// TIA Portal V20 export
ORGANIZATION_BLOCK "Startup"   // OB1015, LAD, Startup
TITLE = "Complete Restart"
// stored: AutoNumber false, IsIECCheckEnabled true, Namespace Unit1.Em2, SetENOAutomatically true
   VAR_INPUT
      LostRetentive : Bool;   // True if retentive data are lost
      LostRTC : Bool;   // True if date and time are lost
   END_VAR
BEGIN

REGION Network 1 (SCL): Build the Absolut Reference Designator
   // Set the Absoult Reference Designator in the Config DB
   IF LEN(IN := "Unit1.Em2.Config".em.referenceDesignator.parent) <> 0 THEN
       "Unit1.Em2.Config".em.referenceDesignator.combined := CONCAT_WSTRING(IN1 := "Unit1.Em2.Config".em.referenceDesignator.parent, IN2 := WSTRING#'.', IN3 := "Unit1.Em2.Config".em.referenceDesignator.relative);
   ELSE
       "Unit1.Em2.Config".em.referenceDesignator.combined := "Unit1.Em2.Config".em.referenceDesignator.relative;
   END_IF;
END_REGION

REGION Network 2 (SCL): CM Config
   // 
   "Unit1.Em2.Config".cmElectrodeFixRightTopFwdBwd .referenceDesignator := WSTRING#'Electrode Fix Right Top';
   "Unit1.Em2.Config".cmElectrodeFixRightTopFwdBwd .monitoringLeavingFeedback := T#5s;
   "Unit1.Em2.Config".cmElectrodeFixRightTopFwdBwd .monitoringReachingFeedback := T#5s;
   "Unit1.Em2.Config".cmElectrodeFixRightTopFwdBwd .monitoringDiscrepancy := T#1s;
   "Unit1.Em2.Config".cmElectrodeFixRightTopFwdBwd .setOutputHomeContinuously := TRUE;
   "Unit1.Em2.Config".cmElectrodeFixRightTopFwdBwd .setOutputWorkContinuously := TRUE;
   "Unit1.Em2.Config".cmElectrodeFixRightTopFwdBwd .disableHomeCommand := FALSE;
   "Unit1.Em2.Config".cmElectrodeFixRightTopFwdBwd .disableFeedbackHomePos := FALSE;
   "Unit1.Em2.Config".cmElectrodeFixRightTopFwdBwd .disableFeedbackWorkPos := FALSE;
   "Unit1.Em2.Config".cmElectrodeFixRightTopFwdBwd .disableAlarms := FALSE;
   "Unit1.Em2.Config".cmElectrodeFixRightTopFwdBwd .resetOutputsOnError := FALSE;
   "Unit1.Em2.Config".cmElectrodeFixRightTopFwdBwd .allwaysWaitOnReachingTime := FALSE;


   // 
   "Unit1.Em2.Config".cmElectrodeFixRightBottomFwdBwd.referenceDesignator := WSTRING#'Electrode Fix Right BTM';
   "Unit1.Em2.Config".cmElectrodeFixRightBottomFwdBwd.monitoringLeavingFeedback := T#5s;
   "Unit1.Em2.Config".cmElectrodeFixRightBottomFwdBwd.monitoringReachingFeedback := T#5s;
   "Unit1.Em2.Config".cmElectrodeFixRightBottomFwdBwd.monitoringDiscrepancy := T#1s;
   "Unit1.Em2.Config".cmElectrodeFixRightBottomFwdBwd.setOutputHomeContinuously := TRUE;
   "Unit1.Em2.Config".cmElectrodeFixRightBottomFwdBwd.setOutputWorkContinuously := TRUE;
   "Unit1.Em2.Config".cmElectrodeFixRightBottomFwdBwd.disableHomeCommand := FALSE;
   "Unit1.Em2.Config".cmElectrodeFixRightBottomFwdBwd.disableFeedbackHomePos := FALSE;
   "Unit1.Em2.Config".cmElectrodeFixRightBottomFwdBwd.disableFeedbackWorkPos := FALSE;
   "Unit1.Em2.Config".cmElectrodeFixRightBottomFwdBwd.disableAlarms := FALSE;
   "Unit1.Em2.Config".cmElectrodeFixRightBottomFwdBwd.resetOutputsOnError := FALSE;
   "Unit1.Em2.Config".cmElectrodeFixRightBottomFwdBwd.allwaysWaitOnReachingTime := FALSE;

   // 
   "Unit1.Em2.Config".cmElectrodeFixLeftTopFwdBwd.referenceDesignator := WSTRING#'Electrode Fix Left Top';
   "Unit1.Em2.Config".cmElectrodeFixLeftTopFwdBwd.monitoringLeavingFeedback := T#5s;
   "Unit1.Em2.Config".cmElectrodeFixLeftTopFwdBwd.monitoringReachingFeedback := T#5s;
   "Unit1.Em2.Config".cmElectrodeFixLeftTopFwdBwd.monitoringDiscrepancy := T#1s;
   "Unit1.Em2.Config".cmElectrodeFixLeftTopFwdBwd.setOutputHomeContinuously := TRUE;
   "Unit1.Em2.Config".cmElectrodeFixLeftTopFwdBwd.setOutputWorkContinuously := TRUE;
   "Unit1.Em2.Config".cmElectrodeFixLeftTopFwdBwd.disableHomeCommand := FALSE;
   "Unit1.Em2.Config".cmElectrodeFixLeftTopFwdBwd.disableFeedbackHomePos := FALSE;
   "Unit1.Em2.Config".cmElectrodeFixLeftTopFwdBwd.disableFeedbackWorkPos := FALSE;
   "Unit1.Em2.Config".cmElectrodeFixLeftTopFwdBwd.disableAlarms := FALSE;
   "Unit1.Em2.Config".cmElectrodeFixLeftTopFwdBwd.resetOutputsOnError := FALSE;
   "Unit1.Em2.Config".cmElectrodeFixLeftTopFwdBwd.allwaysWaitOnReachingTime := FALSE;


   // 
   "Unit1.Em2.Config".cmElectrodeFixLeftBottomFwdBwd.referenceDesignator := WSTRING#'Electrode Fix Left BTM';
   "Unit1.Em2.Config".cmElectrodeFixLeftBottomFwdBwd.monitoringLeavingFeedback := T#5s;
   "Unit1.Em2.Config".cmElectrodeFixLeftBottomFwdBwd.monitoringReachingFeedback := T#5s;
   "Unit1.Em2.Config".cmElectrodeFixLeftBottomFwdBwd.monitoringDiscrepancy := T#1s;
   "Unit1.Em2.Config".cmElectrodeFixLeftBottomFwdBwd.setOutputHomeContinuously := TRUE;
   "Unit1.Em2.Config".cmElectrodeFixLeftBottomFwdBwd.setOutputWorkContinuously := TRUE;
   "Unit1.Em2.Config".cmElectrodeFixLeftBottomFwdBwd.disableHomeCommand := FALSE;
   "Unit1.Em2.Config".cmElectrodeFixLeftBottomFwdBwd.disableFeedbackHomePos := FALSE;
   "Unit1.Em2.Config".cmElectrodeFixLeftBottomFwdBwd.disableFeedbackWorkPos := FALSE;
   "Unit1.Em2.Config".cmElectrodeFixLeftBottomFwdBwd.disableAlarms := FALSE;
   "Unit1.Em2.Config".cmElectrodeFixLeftBottomFwdBwd.resetOutputsOnError := FALSE;
   "Unit1.Em2.Config".cmElectrodeFixLeftBottomFwdBwd.allwaysWaitOnReachingTime := FALSE;


   // 
   "Unit1.Em2.Config".cmElectrodeFixLeftTopUpDown.referenceDesignator := WSTRING#'Electrode Fix Left Top';
   "Unit1.Em2.Config".cmElectrodeFixLeftTopUpDown.monitoringLeavingFeedback := T#5s;
   "Unit1.Em2.Config".cmElectrodeFixLeftTopUpDown.monitoringReachingFeedback := T#5s;
   "Unit1.Em2.Config".cmElectrodeFixLeftTopUpDown.monitoringDiscrepancy := T#1s;
   "Unit1.Em2.Config".cmElectrodeFixLeftTopUpDown.setOutputHomeContinuously := TRUE;
   "Unit1.Em2.Config".cmElectrodeFixLeftTopUpDown.setOutputWorkContinuously := TRUE;
   "Unit1.Em2.Config".cmElectrodeFixLeftTopUpDown.disableHomeCommand := FALSE;
   "Unit1.Em2.Config".cmElectrodeFixLeftTopUpDown.disableFeedbackHomePos := FALSE;
   "Unit1.Em2.Config".cmElectrodeFixLeftTopUpDown.disableFeedbackWorkPos := FALSE;
   "Unit1.Em2.Config".cmElectrodeFixLeftTopUpDown.disableAlarms := FALSE;
   "Unit1.Em2.Config".cmElectrodeFixLeftTopUpDown.resetOutputsOnError := FALSE;
   "Unit1.Em2.Config".cmElectrodeFixLeftTopUpDown.allwaysWaitOnReachingTime := FALSE;


   // 
   "Unit1.Em2.Config".cmElectrodeFixLeftBottomUpDown.referenceDesignator := WSTRING#'Electrode Fix Left BTM';
   "Unit1.Em2.Config".cmElectrodeFixLeftBottomUpDown.monitoringLeavingFeedback := T#5s;
   "Unit1.Em2.Config".cmElectrodeFixLeftBottomUpDown.monitoringReachingFeedback := T#5s;
   "Unit1.Em2.Config".cmElectrodeFixLeftBottomUpDown.monitoringDiscrepancy := T#1s;
   "Unit1.Em2.Config".cmElectrodeFixLeftBottomUpDown.setOutputHomeContinuously := TRUE;
   "Unit1.Em2.Config".cmElectrodeFixLeftBottomUpDown.setOutputWorkContinuously := TRUE;
   "Unit1.Em2.Config".cmElectrodeFixLeftBottomUpDown.disableHomeCommand := FALSE;
   "Unit1.Em2.Config".cmElectrodeFixLeftBottomUpDown.disableFeedbackHomePos := FALSE;
   "Unit1.Em2.Config".cmElectrodeFixLeftBottomUpDown.disableFeedbackWorkPos := FALSE;
   "Unit1.Em2.Config".cmElectrodeFixLeftBottomUpDown.disableAlarms := FALSE;
   "Unit1.Em2.Config".cmElectrodeFixLeftBottomUpDown.resetOutputsOnError := FALSE;
   "Unit1.Em2.Config".cmElectrodeFixLeftBottomUpDown.allwaysWaitOnReachingTime := FALSE;


   // 
   "Unit1.Em2.Config".cmUwSemiSplicerVacuumRightTopOnOff.referenceDesignator := WSTRING#'Splicer Vacuum Right Top';
   "Unit1.Em2.Config".cmUwSemiSplicerVacuumRightTopOnOff.monitoringLeavingFeedback := T#5s;
   "Unit1.Em2.Config".cmUwSemiSplicerVacuumRightTopOnOff.monitoringReachingFeedback := T#1S;
   "Unit1.Em2.Config".cmUwSemiSplicerVacuumRightTopOnOff.monitoringDiscrepancy := T#1s;
   "Unit1.Em2.Config".cmUwSemiSplicerVacuumRightTopOnOff.setOutputHomeContinuously := FALSE;
   "Unit1.Em2.Config".cmUwSemiSplicerVacuumRightTopOnOff.setOutputWorkContinuously := TRUE;
   "Unit1.Em2.Config".cmUwSemiSplicerVacuumRightTopOnOff.disableHomeCommand := FALSE;
   "Unit1.Em2.Config".cmUwSemiSplicerVacuumRightTopOnOff.disableFeedbackHomePos := TRUE;
   "Unit1.Em2.Config".cmUwSemiSplicerVacuumRightTopOnOff.disableFeedbackWorkPos := FALSE;
   "Unit1.Em2.Config".cmUwSemiSplicerVacuumRightTopOnOff.disableAlarms := FALSE;
   "Unit1.Em2.Config".cmUwSemiSplicerVacuumRightTopOnOff.resetOutputsOnError := FALSE;
   "Unit1.Em2.Config".cmUwSemiSplicerVacuumRightTopOnOff.allwaysWaitOnReachingTime := FALSE;


   // 
   "Unit1.Em2.Config".cmUwSemiSplicerVacuumRightBottomOnOff.referenceDesignator := WSTRING#'Splicer Vacuum Right BTM';
   "Unit1.Em2.Config".cmUwSemiSplicerVacuumRightBottomOnOff.monitoringLeavingFeedback := T#5s;
   "Unit1.Em2.Config".cmUwSemiSplicerVacuumRightBottomOnOff.monitoringReachingFeedback := T#1S;
   "Unit1.Em2.Config".cmUwSemiSplicerVacuumRightBottomOnOff.monitoringDiscrepancy := T#1s;
   "Unit1.Em2.Config".cmUwSemiSplicerVacuumRightBottomOnOff.setOutputHomeContinuously := FALSE;
   "Unit1.Em2.Config".cmUwSemiSplicerVacuumRightBottomOnOff.setOutputWorkContinuously := TRUE;
   "Unit1.Em2.Config".cmUwSemiSplicerVacuumRightBottomOnOff.disableHomeCommand := FALSE;
   "Unit1.Em2.Config".cmUwSemiSplicerVacuumRightBottomOnOff.disableFeedbackHomePos := TRUE;
   "Unit1.Em2.Config".cmUwSemiSplicerVacuumRightBottomOnOff.disableFeedbackWorkPos := FALSE;
   "Unit1.Em2.Config".cmUwSemiSplicerVacuumRightBottomOnOff.disableAlarms := FALSE;
   "Unit1.Em2.Config".cmUwSemiSplicerVacuumRightBottomOnOff.resetOutputsOnError := FALSE;
   "Unit1.Em2.Config".cmUwSemiSplicerVacuumRightBottomOnOff.allwaysWaitOnReachingTime := FALSE;


   // 
   "Unit1.Em2.Config".cmUwSemiSplicerVacuumLeftTopOnOff.referenceDesignator := WSTRING#'Splicer Vacuum Left Top';
   "Unit1.Em2.Config".cmUwSemiSplicerVacuumLeftTopOnOff.monitoringLeavingFeedback := T#5s;
   "Unit1.Em2.Config".cmUwSemiSplicerVacuumLeftTopOnOff.monitoringReachingFeedback := T#1S;
   "Unit1.Em2.Config".cmUwSemiSplicerVacuumLeftTopOnOff.monitoringDiscrepancy := T#1s;
   "Unit1.Em2.Config".cmUwSemiSplicerVacuumLeftTopOnOff.setOutputHomeContinuously := FALSE;
   "Unit1.Em2.Config".cmUwSemiSplicerVacuumLeftTopOnOff.setOutputWorkContinuously := TRUE;
   "Unit1.Em2.Config".cmUwSemiSplicerVacuumLeftTopOnOff.disableHomeCommand := FALSE;
   "Unit1.Em2.Config".cmUwSemiSplicerVacuumLeftTopOnOff.disableFeedbackHomePos := TRUE;
   "Unit1.Em2.Config".cmUwSemiSplicerVacuumLeftTopOnOff.disableFeedbackWorkPos := FALSE;
   "Unit1.Em2.Config".cmUwSemiSplicerVacuumLeftTopOnOff.disableAlarms := FALSE;
   "Unit1.Em2.Config".cmUwSemiSplicerVacuumLeftTopOnOff.resetOutputsOnError := FALSE;
   "Unit1.Em2.Config".cmUwSemiSplicerVacuumLeftTopOnOff.allwaysWaitOnReachingTime := FALSE;


   // 
   "Unit1.Em2.Config".cmUwSemiSplicerVacuumLeftBottomOnOff.referenceDesignator := WSTRING#'Splicer Vacuum Left BTM';
   "Unit1.Em2.Config".cmUwSemiSplicerVacuumLeftBottomOnOff.monitoringLeavingFeedback := T#5s;
   "Unit1.Em2.Config".cmUwSemiSplicerVacuumLeftBottomOnOff.monitoringReachingFeedback := T#1S;
   "Unit1.Em2.Config".cmUwSemiSplicerVacuumLeftBottomOnOff.monitoringDiscrepancy := T#1s;
   "Unit1.Em2.Config".cmUwSemiSplicerVacuumLeftBottomOnOff.setOutputHomeContinuously := FALSE;
   "Unit1.Em2.Config".cmUwSemiSplicerVacuumLeftBottomOnOff.setOutputWorkContinuously := TRUE;
   "Unit1.Em2.Config".cmUwSemiSplicerVacuumLeftBottomOnOff.disableHomeCommand := FALSE;
   "Unit1.Em2.Config".cmUwSemiSplicerVacuumLeftBottomOnOff.disableFeedbackHomePos := TRUE;
   "Unit1.Em2.Config".cmUwSemiSplicerVacuumLeftBottomOnOff.disableFeedbackWorkPos := FALSE;
   "Unit1.Em2.Config".cmUwSemiSplicerVacuumLeftBottomOnOff.disableAlarms := FALSE;
   "Unit1.Em2.Config".cmUwSemiSplicerVacuumLeftBottomOnOff.resetOutputsOnError := FALSE;
   "Unit1.Em2.Config".cmUwSemiSplicerVacuumLeftBottomOnOff.allwaysWaitOnReachingTime := FALSE;


   // Electrode Cutter
   "Unit1.Em2.Config".cmElectrodeCutterFwdBwd.referenceDesignator := WSTRING#'Electrode Cutter';
   "Unit1.Em2.Config".cmElectrodeCutterFwdBwd.monitoringLeavingFeedback := T#5s;
   "Unit1.Em2.Config".cmElectrodeCutterFwdBwd.monitoringReachingFeedback := T#5s;
   "Unit1.Em2.Config".cmElectrodeCutterFwdBwd.monitoringDiscrepancy := T#1s;
   "Unit1.Em2.Config".cmElectrodeCutterFwdBwd.setOutputHomeContinuously := TRUE;
   "Unit1.Em2.Config".cmElectrodeCutterFwdBwd.setOutputWorkContinuously := TRUE;
   "Unit1.Em2.Config".cmElectrodeCutterFwdBwd.disableHomeCommand := FALSE;
   "Unit1.Em2.Config".cmElectrodeCutterFwdBwd.disableFeedbackHomePos := FALSE;
   "Unit1.Em2.Config".cmElectrodeCutterFwdBwd.disableFeedbackWorkPos := FALSE;
   "Unit1.Em2.Config".cmElectrodeCutterFwdBwd.disableAlarms := FALSE;
   "Unit1.Em2.Config".cmElectrodeCutterFwdBwd.resetOutputsOnError := FALSE;
   "Unit1.Em2.Config".cmElectrodeCutterFwdBwd.allwaysWaitOnReachingTime := FALSE;


   // 
   "Unit1.Em2.Config".cmSplicingLeftModuleMoverFwdBwd.referenceDesignator := WSTRING#'Left Module Mover';
   "Unit1.Em2.Config".cmSplicingLeftModuleMoverFwdBwd.monitoringLeavingFeedback := T#30s;
   "Unit1.Em2.Config".cmSplicingLeftModuleMoverFwdBwd.monitoringReachingFeedback := T#30s;
   "Unit1.Em2.Config".cmSplicingLeftModuleMoverFwdBwd.monitoringDiscrepancy := T#1s;
   "Unit1.Em2.Config".cmSplicingLeftModuleMoverFwdBwd.setOutputHomeContinuously := TRUE;
   "Unit1.Em2.Config".cmSplicingLeftModuleMoverFwdBwd.setOutputWorkContinuously := TRUE;
   "Unit1.Em2.Config".cmSplicingLeftModuleMoverFwdBwd.disableHomeCommand := FALSE;
   "Unit1.Em2.Config".cmSplicingLeftModuleMoverFwdBwd.disableFeedbackHomePos := FALSE;
   "Unit1.Em2.Config".cmSplicingLeftModuleMoverFwdBwd.disableFeedbackWorkPos := FALSE;
   "Unit1.Em2.Config".cmSplicingLeftModuleMoverFwdBwd.disableAlarms := FALSE;
   "Unit1.Em2.Config".cmSplicingLeftModuleMoverFwdBwd.resetOutputsOnError := FALSE;
   "Unit1.Em2.Config".cmSplicingLeftModuleMoverFwdBwd.allwaysWaitOnReachingTime := FALSE;


   // 
   "Unit1.Em2.Config".cmSplicingRightModuleMoverFwdBwd.referenceDesignator := WSTRING#'Right Module Mover';
   "Unit1.Em2.Config".cmSplicingRightModuleMoverFwdBwd.monitoringLeavingFeedback := T#30s;
   "Unit1.Em2.Config".cmSplicingRightModuleMoverFwdBwd.monitoringReachingFeedback := T#30s;
   "Unit1.Em2.Config".cmSplicingRightModuleMoverFwdBwd.monitoringDiscrepancy := T#1s;
   "Unit1.Em2.Config".cmSplicingRightModuleMoverFwdBwd.setOutputHomeContinuously := TRUE;
   "Unit1.Em2.Config".cmSplicingRightModuleMoverFwdBwd.setOutputWorkContinuously := TRUE;
   "Unit1.Em2.Config".cmSplicingRightModuleMoverFwdBwd.disableHomeCommand := FALSE;
   "Unit1.Em2.Config".cmSplicingRightModuleMoverFwdBwd.disableFeedbackHomePos := FALSE;
   "Unit1.Em2.Config".cmSplicingRightModuleMoverFwdBwd.disableFeedbackWorkPos := FALSE;
   "Unit1.Em2.Config".cmSplicingRightModuleMoverFwdBwd.disableAlarms := FALSE;
   "Unit1.Em2.Config".cmSplicingRightModuleMoverFwdBwd.resetOutputsOnError := FALSE;
   "Unit1.Em2.Config".cmSplicingRightModuleMoverFwdBwd.allwaysWaitOnReachingTime := FALSE;


   // 
   "Unit1.Em2.Config".cmElectrodeLeftHolderMoverFwdBwd.referenceDesignator := WSTRING#'Left Holder Mover';
   "Unit1.Em2.Config".cmElectrodeLeftHolderMoverFwdBwd.monitoringLeavingFeedback := T#5s;
   "Unit1.Em2.Config".cmElectrodeLeftHolderMoverFwdBwd.monitoringReachingFeedback := T#5s;
   "Unit1.Em2.Config".cmElectrodeLeftHolderMoverFwdBwd.monitoringDiscrepancy := T#1s;
   "Unit1.Em2.Config".cmElectrodeLeftHolderMoverFwdBwd.setOutputHomeContinuously := TRUE;
   "Unit1.Em2.Config".cmElectrodeLeftHolderMoverFwdBwd.setOutputWorkContinuously := TRUE;
   "Unit1.Em2.Config".cmElectrodeLeftHolderMoverFwdBwd.disableHomeCommand := FALSE;
   "Unit1.Em2.Config".cmElectrodeLeftHolderMoverFwdBwd.disableFeedbackHomePos := FALSE;
   "Unit1.Em2.Config".cmElectrodeLeftHolderMoverFwdBwd.disableFeedbackWorkPos := FALSE;
   "Unit1.Em2.Config".cmElectrodeLeftHolderMoverFwdBwd.disableAlarms := FALSE;
   "Unit1.Em2.Config".cmElectrodeLeftHolderMoverFwdBwd.resetOutputsOnError := FALSE;
   "Unit1.Em2.Config".cmElectrodeLeftHolderMoverFwdBwd.allwaysWaitOnReachingTime := FALSE;


   // 
   "Unit1.Em2.Config".cmElectrodeRightHolderMoverFwdBwd.referenceDesignator := WSTRING#'Right Holder Mover';
   "Unit1.Em2.Config".cmElectrodeRightHolderMoverFwdBwd.monitoringLeavingFeedback := T#5s;
   "Unit1.Em2.Config".cmElectrodeRightHolderMoverFwdBwd.monitoringReachingFeedback := T#5s;
   "Unit1.Em2.Config".cmElectrodeRightHolderMoverFwdBwd.monitoringDiscrepancy := T#1s;
   "Unit1.Em2.Config".cmElectrodeRightHolderMoverFwdBwd.setOutputHomeContinuously := TRUE;
   "Unit1.Em2.Config".cmElectrodeRightHolderMoverFwdBwd.setOutputWorkContinuously := TRUE;
   "Unit1.Em2.Config".cmElectrodeRightHolderMoverFwdBwd.disableHomeCommand := FALSE;
   "Unit1.Em2.Config".cmElectrodeRightHolderMoverFwdBwd.disableFeedbackHomePos := FALSE;
   "Unit1.Em2.Config".cmElectrodeRightHolderMoverFwdBwd.disableFeedbackWorkPos := FALSE;
   "Unit1.Em2.Config".cmElectrodeRightHolderMoverFwdBwd.disableAlarms := FALSE;
   "Unit1.Em2.Config".cmElectrodeRightHolderMoverFwdBwd.resetOutputsOnError := FALSE;
   "Unit1.Em2.Config".cmElectrodeRightHolderMoverFwdBwd.allwaysWaitOnReachingTime := FALSE;


   // Tape Loading Turn Table
   "Unit1.Em2.Config".cmTapeLoadingTurnCwCcw.referenceDesignator := WSTRING#'Tape Loading Tum';
   "Unit1.Em2.Config".cmTapeLoadingTurnCwCcw.monitoringLeavingFeedback := T#5s;
   "Unit1.Em2.Config".cmTapeLoadingTurnCwCcw.monitoringReachingFeedback := T#5s;
   "Unit1.Em2.Config".cmTapeLoadingTurnCwCcw.monitoringDiscrepancy := T#1s;
   "Unit1.Em2.Config".cmTapeLoadingTurnCwCcw.setOutputHomeContinuously := TRUE;
   "Unit1.Em2.Config".cmTapeLoadingTurnCwCcw.setOutputWorkContinuously := TRUE;
   "Unit1.Em2.Config".cmTapeLoadingTurnCwCcw.disableHomeCommand := FALSE;
   "Unit1.Em2.Config".cmTapeLoadingTurnCwCcw.disableFeedbackHomePos := FALSE;
   "Unit1.Em2.Config".cmTapeLoadingTurnCwCcw.disableFeedbackWorkPos := FALSE;
   "Unit1.Em2.Config".cmTapeLoadingTurnCwCcw.disableAlarms := FALSE;
   "Unit1.Em2.Config".cmTapeLoadingTurnCwCcw.resetOutputsOnError := FALSE;
   "Unit1.Em2.Config".cmTapeLoadingTurnCwCcw.allwaysWaitOnReachingTime := FALSE;


   // Tape Attach Unit
   "Unit1.Em2.Config".cmTapeAttachUnitFwdBwd.referenceDesignator := WSTRING#'Tape Attach Unit';
   "Unit1.Em2.Config".cmTapeAttachUnitFwdBwd.monitoringLeavingFeedback := T#5s;
   "Unit1.Em2.Config".cmTapeAttachUnitFwdBwd.monitoringReachingFeedback := T#5s;
   "Unit1.Em2.Config".cmTapeAttachUnitFwdBwd.monitoringDiscrepancy := T#1s;
   "Unit1.Em2.Config".cmTapeAttachUnitFwdBwd.setOutputHomeContinuously := TRUE;
   "Unit1.Em2.Config".cmTapeAttachUnitFwdBwd.setOutputWorkContinuously := TRUE;
   "Unit1.Em2.Config".cmTapeAttachUnitFwdBwd.disableHomeCommand := FALSE;
   "Unit1.Em2.Config".cmTapeAttachUnitFwdBwd.disableFeedbackHomePos := FALSE;
   "Unit1.Em2.Config".cmTapeAttachUnitFwdBwd.disableFeedbackWorkPos := FALSE;
   "Unit1.Em2.Config".cmTapeAttachUnitFwdBwd.disableAlarms := FALSE;
   "Unit1.Em2.Config".cmTapeAttachUnitFwdBwd.resetOutputsOnError := FALSE;
   "Unit1.Em2.Config".cmTapeAttachUnitFwdBwd.allwaysWaitOnReachingTime := FALSE;


   // Tape Vacuum
   "Unit1.Em2.Config".cmTapeVacuumOnOff.referenceDesignator := WSTRING#'Tape Vacuum';
   "Unit1.Em2.Config".cmTapeVacuumOnOff.monitoringLeavingFeedback := T#5s;
   "Unit1.Em2.Config".cmTapeVacuumOnOff.monitoringReachingFeedback := T#1s;
   "Unit1.Em2.Config".cmTapeVacuumOnOff.monitoringDiscrepancy := T#1s;
   "Unit1.Em2.Config".cmTapeVacuumOnOff.setOutputHomeContinuously := FALSE;
   "Unit1.Em2.Config".cmTapeVacuumOnOff.setOutputWorkContinuously := TRUE;
   "Unit1.Em2.Config".cmTapeVacuumOnOff.disableHomeCommand := FALSE;
   "Unit1.Em2.Config".cmTapeVacuumOnOff.disableFeedbackHomePos := TRUE;
   "Unit1.Em2.Config".cmTapeVacuumOnOff.disableFeedbackWorkPos := FALSE;
   "Unit1.Em2.Config".cmTapeVacuumOnOff.disableAlarms := FALSE;
   "Unit1.Em2.Config".cmTapeVacuumOnOff.resetOutputsOnError := FALSE;
   "Unit1.Em2.Config".cmTapeVacuumOnOff.allwaysWaitOnReachingTime := FALSE;


   // Stopper
   "Unit1.Em2.Config".cmStopperFwdBwd.referenceDesignator := WSTRING#'Stopper';
   "Unit1.Em2.Config".cmStopperFwdBwd.monitoringLeavingFeedback := T#5s;
   "Unit1.Em2.Config".cmStopperFwdBwd.monitoringReachingFeedback := T#5s;
   "Unit1.Em2.Config".cmStopperFwdBwd.monitoringDiscrepancy := T#1s;
   "Unit1.Em2.Config".cmStopperFwdBwd.setOutputHomeContinuously := TRUE;
   "Unit1.Em2.Config".cmStopperFwdBwd.setOutputWorkContinuously := TRUE;
   "Unit1.Em2.Config".cmStopperFwdBwd.disableHomeCommand := FALSE;
   "Unit1.Em2.Config".cmStopperFwdBwd.disableFeedbackHomePos := FALSE;
   "Unit1.Em2.Config".cmStopperFwdBwd.disableFeedbackWorkPos := FALSE;
   "Unit1.Em2.Config".cmStopperFwdBwd.disableAlarms := FALSE;
   "Unit1.Em2.Config".cmStopperFwdBwd.resetOutputsOnError := FALSE;
   "Unit1.Em2.Config".cmStopperFwdBwd.allwaysWaitOnReachingTime := FALSE;


   // Support Unit Transfer
   "Unit1.Em2.Config".cmSupportUnitTransferFwdBwd.referenceDesignator := WSTRING#'Support Unit Transfer';
   "Unit1.Em2.Config".cmSupportUnitTransferFwdBwd.monitoringLeavingFeedback := T#30s;
   "Unit1.Em2.Config".cmSupportUnitTransferFwdBwd.monitoringReachingFeedback := T#30s;
   "Unit1.Em2.Config".cmSupportUnitTransferFwdBwd.monitoringDiscrepancy := T#1s;
   "Unit1.Em2.Config".cmSupportUnitTransferFwdBwd.setOutputHomeContinuously := TRUE;
   "Unit1.Em2.Config".cmSupportUnitTransferFwdBwd.setOutputWorkContinuously := TRUE;
   "Unit1.Em2.Config".cmSupportUnitTransferFwdBwd.disableHomeCommand := FALSE;
   "Unit1.Em2.Config".cmSupportUnitTransferFwdBwd.disableFeedbackHomePos := FALSE;
   "Unit1.Em2.Config".cmSupportUnitTransferFwdBwd.disableFeedbackWorkPos := FALSE;
   "Unit1.Em2.Config".cmSupportUnitTransferFwdBwd.disableAlarms := FALSE;
   "Unit1.Em2.Config".cmSupportUnitTransferFwdBwd.resetOutputsOnError := FALSE;
   "Unit1.Em2.Config".cmSupportUnitTransferFwdBwd.allwaysWaitOnReachingTime := FALSE;


   // Support Unit Shaft
   "Unit1.Em2.Config".cmSupportUnitShaftUpDown.referenceDesignator := WSTRING#'Support Unit Shaft';
   "Unit1.Em2.Config".cmSupportUnitShaftUpDown.monitoringLeavingFeedback := T#5s;
   "Unit1.Em2.Config".cmSupportUnitShaftUpDown.monitoringReachingFeedback := T#5s;
   "Unit1.Em2.Config".cmSupportUnitShaftUpDown.monitoringDiscrepancy := T#1s;
   "Unit1.Em2.Config".cmSupportUnitShaftUpDown.setOutputHomeContinuously := TRUE;
   "Unit1.Em2.Config".cmSupportUnitShaftUpDown.setOutputWorkContinuously := TRUE;
   "Unit1.Em2.Config".cmSupportUnitShaftUpDown.disableHomeCommand := FALSE;
   "Unit1.Em2.Config".cmSupportUnitShaftUpDown.disableFeedbackHomePos := FALSE;
   "Unit1.Em2.Config".cmSupportUnitShaftUpDown.disableFeedbackWorkPos := FALSE;
   "Unit1.Em2.Config".cmSupportUnitShaftUpDown.disableAlarms := FALSE;
   "Unit1.Em2.Config".cmSupportUnitShaftUpDown.resetOutputsOnError := FALSE;
   "Unit1.Em2.Config".cmSupportUnitShaftUpDown.allwaysWaitOnReachingTime := FALSE;


   // Frame Cover
   "Unit1.Em2.Config".cmFrameCoverFwdBwd.referenceDesignator := WSTRING#'Frame Cover';
   "Unit1.Em2.Config".cmFrameCoverFwdBwd.monitoringLeavingFeedback := T#5s;
   "Unit1.Em2.Config".cmFrameCoverFwdBwd.monitoringReachingFeedback := T#5s;
   "Unit1.Em2.Config".cmFrameCoverFwdBwd.monitoringDiscrepancy := T#1s;
   "Unit1.Em2.Config".cmFrameCoverFwdBwd.setOutputHomeContinuously := TRUE;
   "Unit1.Em2.Config".cmFrameCoverFwdBwd.setOutputWorkContinuously := TRUE;
   "Unit1.Em2.Config".cmFrameCoverFwdBwd.disableHomeCommand := FALSE;
   "Unit1.Em2.Config".cmFrameCoverFwdBwd.disableFeedbackHomePos := FALSE;
   "Unit1.Em2.Config".cmFrameCoverFwdBwd.disableFeedbackWorkPos := FALSE;
   "Unit1.Em2.Config".cmFrameCoverFwdBwd.disableAlarms := FALSE;
   "Unit1.Em2.Config".cmFrameCoverFwdBwd.resetOutputsOnError := FALSE;
   "Unit1.Em2.Config".cmFrameCoverFwdBwd.allwaysWaitOnReachingTime := FALSE;
END_REGION
END_ORGANIZATION_BLOCK
